PROGRAM pouStation1
VAR
	stationMode: FB_Mode;
	tCalcNumberOfPages: REAL;
	ceil: REAL;
	PartBuild: FB_PartBuild;
	retvall: UDINT;
	
	
	// TODO
	tPartPresent: BOOL;
END_VAR

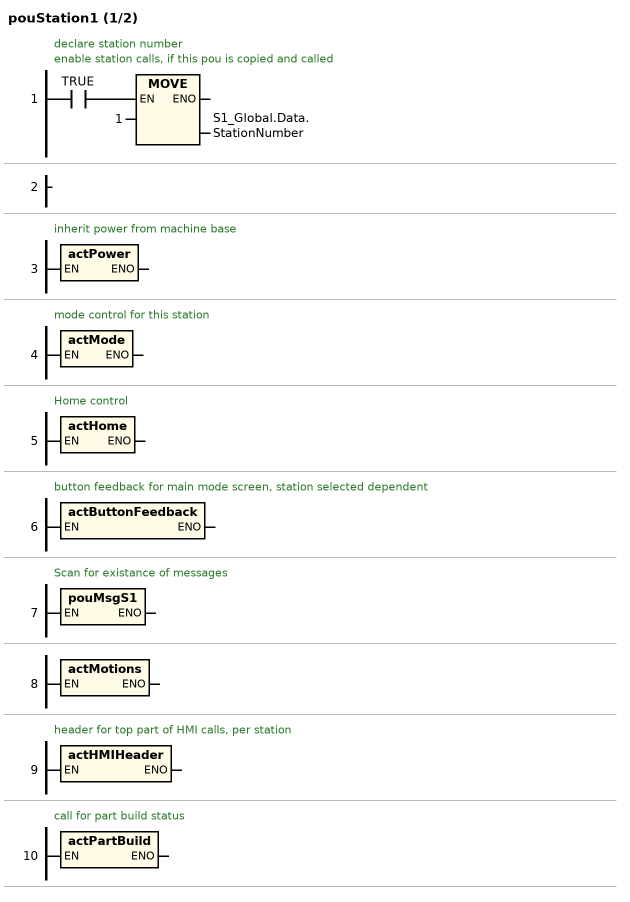
// NETWORK 1
// declare station number
// enable station calls, if this pou is copied and called
S1_Global.Data.StationNumber := 1;

// NETWORK 2

// NETWORK 3
// inherit power from machine base
actPower();

// NETWORK 4
// mode control for this station
actMode();

// NETWORK 5
// Home control
actHome();

// NETWORK 6
// button feedback for main mode screen, station selected dependent
actButtonFeedback();

// NETWORK 7
// Scan for existance of messages
pouMsgS1();

// NETWORK 8
actMotions();

// NETWORK 9
// header for top part of HMI calls, per station
actHMIHeader();

// NETWORK 10
// call for part build status
actPartBuild();

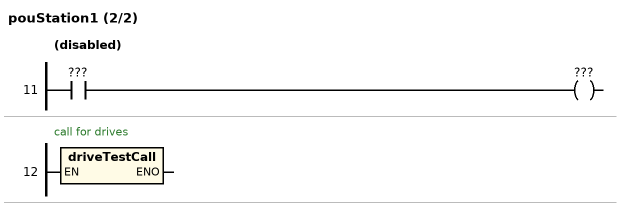
// NETWORK 11 (disabled)
// ??? := ???;

// NETWORK 12
// call for drives
driveTestCall();

ACTION actButtonFeedback:
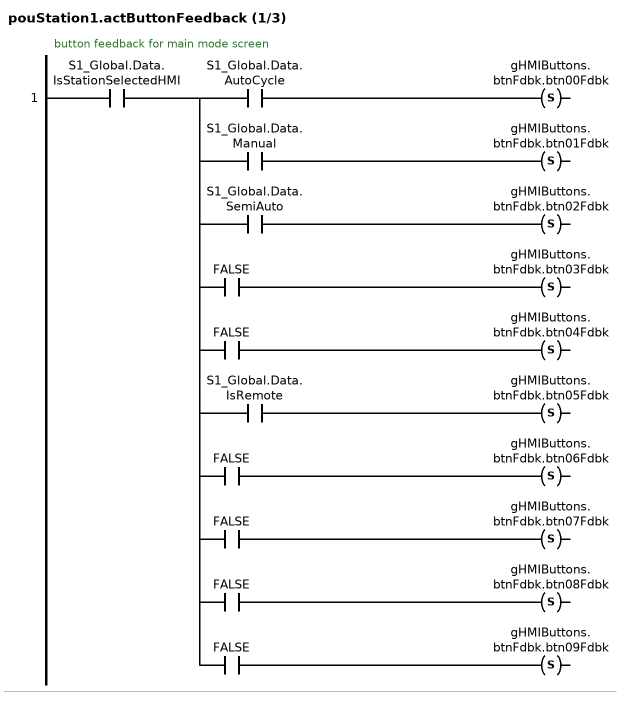
// NETWORK 1
// button feedback for main mode screen
gHMIButtons.btnFdbk.btn00Fdbk S= S1_Global.Data.IsStationSelectedHMI AND S1_Global.Data.AutoCycle;
gHMIButtons.btnFdbk.btn01Fdbk S= S1_Global.Data.IsStationSelectedHMI AND S1_Global.Data.Manual;
gHMIButtons.btnFdbk.btn02Fdbk S= S1_Global.Data.IsStationSelectedHMI AND S1_Global.Data.SemiAuto;
gHMIButtons.btnFdbk.btn03Fdbk S= S1_Global.Data.IsStationSelectedHMI AND FALSE;
gHMIButtons.btnFdbk.btn04Fdbk S= S1_Global.Data.IsStationSelectedHMI AND FALSE;
gHMIButtons.btnFdbk.btn05Fdbk S= S1_Global.Data.IsStationSelectedHMI AND S1_Global.Data.IsRemote;
gHMIButtons.btnFdbk.btn06Fdbk S= S1_Global.Data.IsStationSelectedHMI AND FALSE;
gHMIButtons.btnFdbk.btn07Fdbk S= S1_Global.Data.IsStationSelectedHMI AND FALSE;
gHMIButtons.btnFdbk.btn08Fdbk S= S1_Global.Data.IsStationSelectedHMI AND FALSE;
gHMIButtons.btnFdbk.btn09Fdbk S= S1_Global.Data.IsStationSelectedHMI AND FALSE;

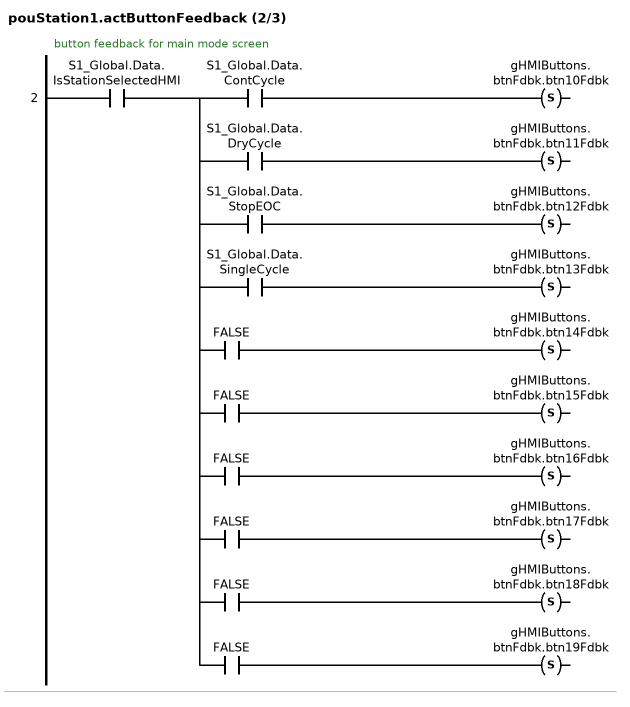
// NETWORK 2
// button feedback for main mode screen
gHMIButtons.btnFdbk.btn10Fdbk S= S1_Global.Data.IsStationSelectedHMI AND S1_Global.Data.ContCycle;
gHMIButtons.btnFdbk.btn11Fdbk S= S1_Global.Data.IsStationSelectedHMI AND S1_Global.Data.DryCycle;
gHMIButtons.btnFdbk.btn12Fdbk S= S1_Global.Data.IsStationSelectedHMI AND S1_Global.Data.StopEOC;
gHMIButtons.btnFdbk.btn13Fdbk S= S1_Global.Data.IsStationSelectedHMI AND S1_Global.Data.SingleCycle;
gHMIButtons.btnFdbk.btn14Fdbk S= S1_Global.Data.IsStationSelectedHMI AND FALSE;
gHMIButtons.btnFdbk.btn15Fdbk S= S1_Global.Data.IsStationSelectedHMI AND FALSE;
gHMIButtons.btnFdbk.btn16Fdbk S= S1_Global.Data.IsStationSelectedHMI AND FALSE;
gHMIButtons.btnFdbk.btn17Fdbk S= S1_Global.Data.IsStationSelectedHMI AND FALSE;
gHMIButtons.btnFdbk.btn18Fdbk S= S1_Global.Data.IsStationSelectedHMI AND FALSE;
gHMIButtons.btnFdbk.btn19Fdbk S= S1_Global.Data.IsStationSelectedHMI AND FALSE;

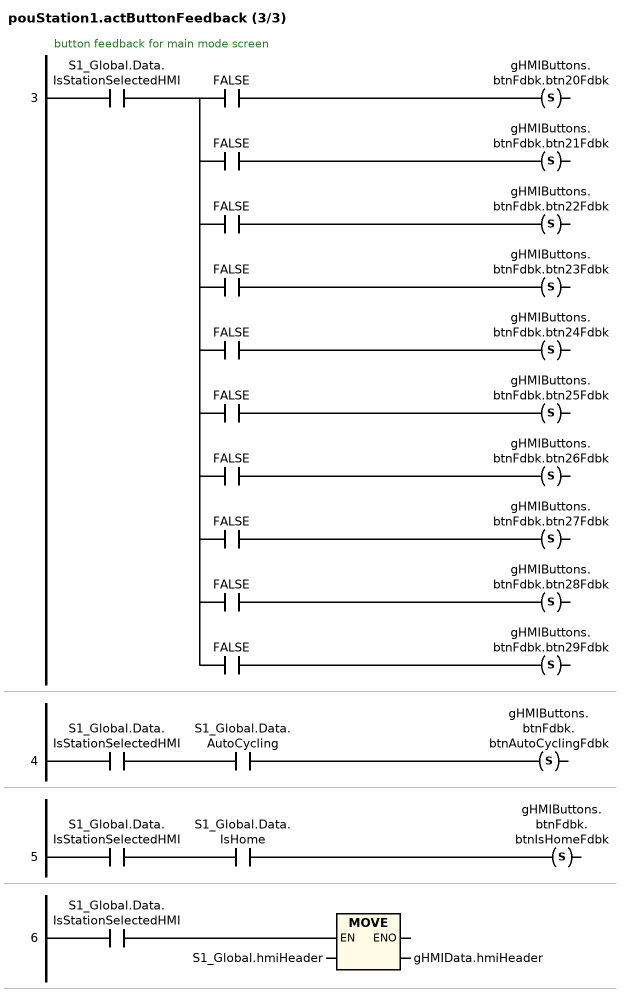
// NETWORK 3
// button feedback for main mode screen
gHMIButtons.btnFdbk.btn20Fdbk S= S1_Global.Data.IsStationSelectedHMI AND FALSE;
gHMIButtons.btnFdbk.btn21Fdbk S= S1_Global.Data.IsStationSelectedHMI AND FALSE;
gHMIButtons.btnFdbk.btn22Fdbk S= S1_Global.Data.IsStationSelectedHMI AND FALSE;
gHMIButtons.btnFdbk.btn23Fdbk S= S1_Global.Data.IsStationSelectedHMI AND FALSE;
gHMIButtons.btnFdbk.btn24Fdbk S= S1_Global.Data.IsStationSelectedHMI AND FALSE;
gHMIButtons.btnFdbk.btn25Fdbk S= S1_Global.Data.IsStationSelectedHMI AND FALSE;
gHMIButtons.btnFdbk.btn26Fdbk S= S1_Global.Data.IsStationSelectedHMI AND FALSE;
gHMIButtons.btnFdbk.btn27Fdbk S= S1_Global.Data.IsStationSelectedHMI AND FALSE;
gHMIButtons.btnFdbk.btn28Fdbk S= S1_Global.Data.IsStationSelectedHMI AND FALSE;
gHMIButtons.btnFdbk.btn29Fdbk S= S1_Global.Data.IsStationSelectedHMI AND FALSE;

// NETWORK 4
gHMIButtons.btnFdbk.btnAutoCyclingFdbk S= S1_Global.Data.IsStationSelectedHMI AND S1_Global.Data.AutoCycling;

// NETWORK 5
gHMIButtons.btnFdbk.btnIsHomeFdbk S= S1_Global.Data.IsStationSelectedHMI AND S1_Global.Data.IsHome;

// NETWORK 6
IF S1_Global.Data.IsStationSelectedHMI THEN gHMIData.hmiHeader := S1_Global.hmiHeader; END_IF
END_ACTION

ACTION actHMIHeader:
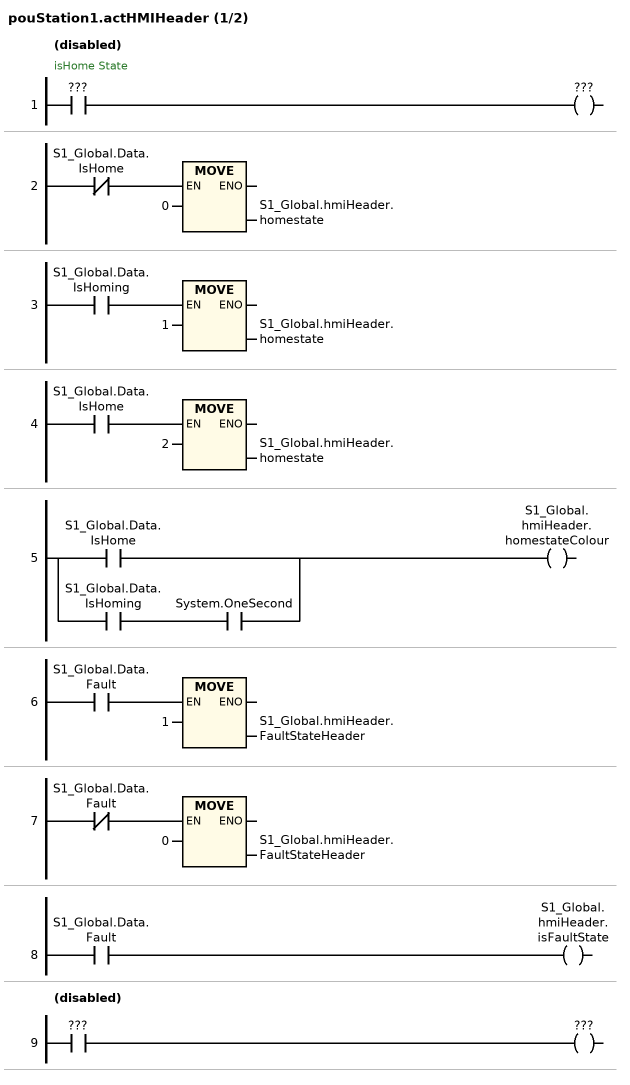
// NETWORK 1 (disabled)
// isHome State
// ??? := ???;

// NETWORK 2
IF NOT S1_Global.Data.IsHome THEN S1_Global.hmiHeader.homestate := 0; END_IF

// NETWORK 3
IF S1_Global.Data.IsHoming THEN S1_Global.hmiHeader.homestate := 1; END_IF

// NETWORK 4
IF S1_Global.Data.IsHome THEN S1_Global.hmiHeader.homestate := 2; END_IF

// NETWORK 5
S1_Global.hmiHeader.homestateColour := S1_Global.Data.IsHome OR S1_Global.Data.IsHoming AND System.OneSecond;

// NETWORK 6
IF S1_Global.Data.Fault THEN S1_Global.hmiHeader.FaultStateHeader := 1; END_IF

// NETWORK 7
IF NOT S1_Global.Data.Fault THEN S1_Global.hmiHeader.FaultStateHeader := 0; END_IF

// NETWORK 8
S1_Global.hmiHeader.isFaultState := S1_Global.Data.Fault;

// NETWORK 9 (disabled)
// ??? := ???;

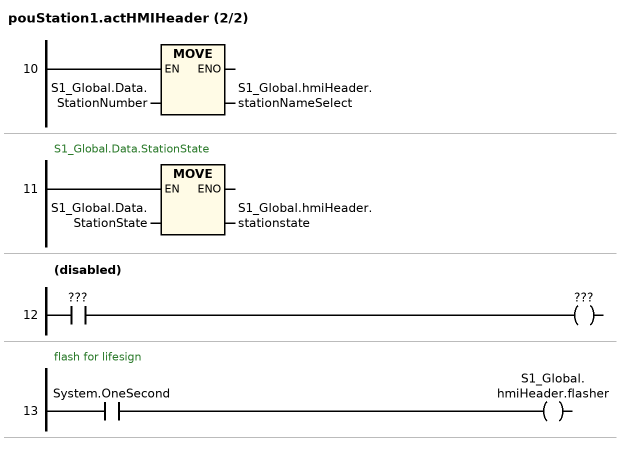
// NETWORK 10
S1_Global.hmiHeader.stationNameSelect := S1_Global.Data.StationNumber;

// NETWORK 11
// S1_Global.Data.StationState
S1_Global.hmiHeader.stationstate := S1_Global.Data.StationState;

// NETWORK 12 (disabled)
// ??? := ???;

// NETWORK 13
// flash for lifesign
S1_Global.hmiHeader.flasher := System.OneSecond;
END_ACTION

ACTION actHome:
//Set home status for station

IF 
//are all motions returned
S1_01_Motion_01_01.Motion.qReturnDepth AND
S1_01_Motion_01_02.Motion.qReturnDepth AND
S1_01_Motion_01_03.Motion.qReturnDepth AND
S1_01_Motion_01_04.Motion.qReturnDepth AND
S1_01_Motion_01_05.Motion.qReturnDepth AND
S1_01_Motion_01_06.Motion.qReturnDepth

	THEN
		//set IsHome value for station
		S1_Global.Data.IsHome := TRUE;
	ELSE
		S1_Global.Data.IsHome := FALSE;
END_IF
END_ACTION

ACTION actMaxNumStationPages:
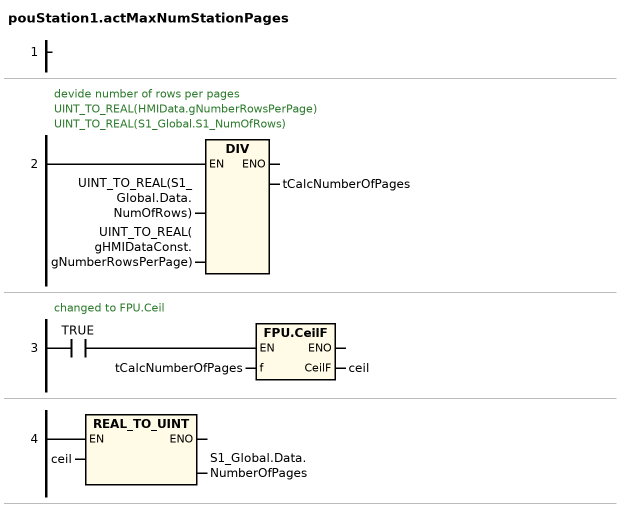
// NETWORK 1

// NETWORK 2
// devide number of rows per pages
// UINT_TO_REAL(HMIData.gNumberRowsPerPage)
// UINT_TO_REAL(S1_Global.S1_NumOfRows)
tCalcNumberOfPages := (UINT_TO_REAL(S1_Global.Data.NumOfRows)) / (UINT_TO_REAL(gHMIDataConst.gNumberRowsPerPage));

// NETWORK 3
// changed to FPU.Ceil
ceil := FPU.CeilF(f := tCalcNumberOfPages);

// NETWORK 4
S1_Global.Data.NumberOfPages := REAL_TO_UINT(ceil);
END_ACTION

ACTION actMode:
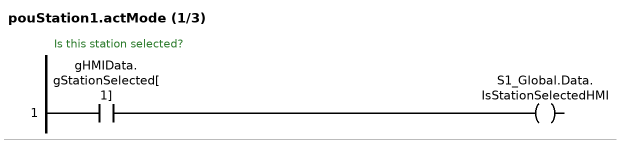
// NETWORK 1
// Is this station selected?
S1_Global.Data.IsStationSelectedHMI := gHMIData.gStationSelected[1];

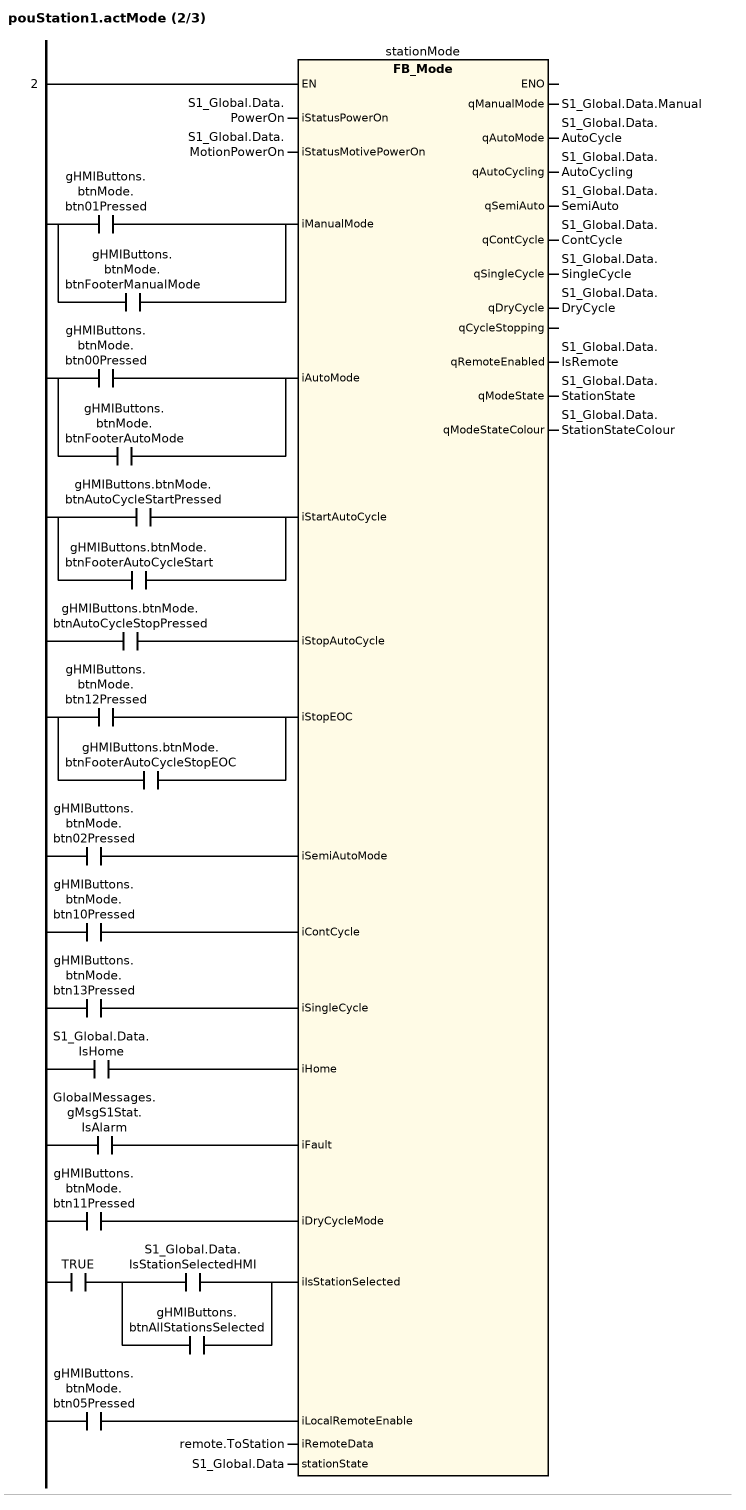
// NETWORK 2
stationMode(
    iStatusPowerOn := S1_Global.Data.PowerOn,
    iStatusMotivePowerOn := S1_Global.Data.MotionPowerOn,
    iManualMode := gHMIButtons.btnMode.btn01Pressed OR gHMIButtons.btnMode.btnFooterManualMode,
    iAutoMode := gHMIButtons.btnMode.btn00Pressed OR gHMIButtons.btnMode.btnFooterAutoMode,
    iStartAutoCycle := gHMIButtons.btnMode.btnAutoCycleStartPressed OR gHMIButtons.btnMode.btnFooterAutoCycleStart,
    iStopAutoCycle := gHMIButtons.btnMode.btnAutoCycleStopPressed,
    iStopEOC := gHMIButtons.btnMode.btn12Pressed OR gHMIButtons.btnMode.btnFooterAutoCycleStopEOC,
    iSemiAutoMode := gHMIButtons.btnMode.btn02Pressed,
    iContCycle := gHMIButtons.btnMode.btn10Pressed,
    iSingleCycle := gHMIButtons.btnMode.btn13Pressed,
    iHome := S1_Global.Data.IsHome,
    iFault := GlobalMessages.gMsgS1Stat.IsAlarm,
    iDryCycleMode := gHMIButtons.btnMode.btn11Pressed,
    iIsStationSelected := TRUE AND (S1_Global.Data.IsStationSelectedHMI OR gHMIButtons.btnAllStationsSelected),
    iLocalRemoteEnable := gHMIButtons.btnMode.btn05Pressed,
    iRemoteData := remote.ToStation,
    stationState := S1_Global.Data,
    qManualMode => S1_Global.Data.Manual,
    qAutoMode => S1_Global.Data.AutoCycle,
    qAutoCycling => S1_Global.Data.AutoCycling,
    qSemiAuto => S1_Global.Data.SemiAuto,
    qContCycle => S1_Global.Data.ContCycle,
    qSingleCycle => S1_Global.Data.SingleCycle,
    qDryCycle => S1_Global.Data.DryCycle,
    qRemoteEnabled => S1_Global.Data.IsRemote,
    qModeState => S1_Global.Data.StationState,
    qModeStateColour => S1_Global.Data.StationStateColour); // FB_Mode

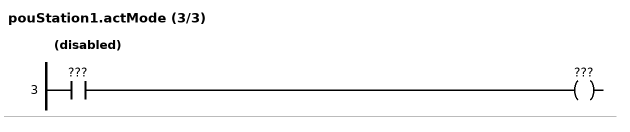
// NETWORK 3 (disabled)
// ??? := ???;
END_ACTION

ACTION actMotions:
//station 1 = 10000 index


//init number of rows
S1_Global.Data.NumOfRows := 0;

//page 1
S1_01_Motion_01_01();
S1_01_Motion_01_02();
S1_01_Motion_01_03();
S1_01_Motion_01_04();
S1_01_Motion_01_05();
S1_01_Motion_01_06();

//page 2
S1_01_Motion_02_07();
S1_01_Motion_02_08();
S1_01_Motion_02_09();
S1_01_Motion_02_10();
S1_01_Motion_02_11();
S1_01_Motion_02_12();

//page 3
S1_01_Motion_03_13();
S1_01_Motion_03_14();
S1_01_Motion_03_15();
S1_01_Motion_03_16();
S1_01_Motion_03_17();
S1_01_Motion_03_18();

//page 4
S1_01_Motion_04_19();
S1_01_Motion_04_20();
S1_01_Motion_04_21();
S1_01_Motion_04_22();
S1_01_Motion_04_23();
S1_01_Motion_04_24();

//page 5
S1_01_Motion_05_25();
S1_01_Motion_05_26();
S1_01_Motion_05_27();
S1_01_Motion_05_28();
S1_01_Motion_05_29();
S1_01_Motion_05_30();

//page 6
S1_01_Motion_06_31();
S1_01_Motion_06_32();
S1_01_Motion_06_33();
S1_01_Motion_06_34();
S1_01_Motion_06_35();
S1_01_Motion_06_36();

//must be called after motionRow calls
actMaxNumStationPages();
END_ACTION

ACTION actPartBuild:
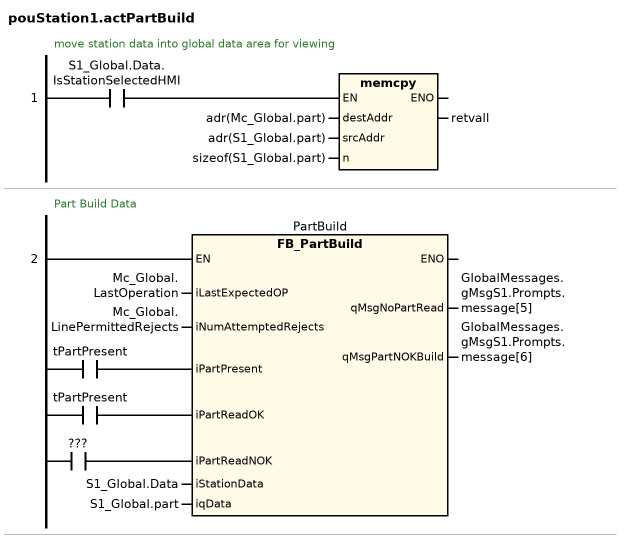
// NETWORK 1
// move station data into global data area for viewing
IF S1_Global.Data.IsStationSelectedHMI THEN
    retvall := memcpy(destAddr := adr(Mc_Global.part), srcAddr := adr(S1_Global.part), n := sizeof(S1_Global.part));
END_IF

// NETWORK 2
// Part Build Data
PartBuild(
    iLastExpectedOP := Mc_Global.LastOperation,
    iNumAttemptedRejects := Mc_Global.LinePermittedRejects,
    iPartPresent := tPartPresent,
    iPartReadOK := tPartPresent,
    iStationData := S1_Global.Data,
    iqData := S1_Global.part,
    qMsgNoPartRead => GlobalMessages.gMsgS1.Prompts.message[5],
    qMsgPartNOKBuild => GlobalMessages.gMsgS1.Prompts.message[6]); // FB_PartBuild
END_ACTION

ACTION actPower:
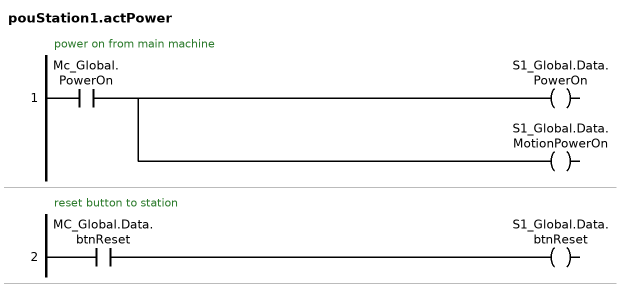
// NETWORK 1
// power on from main machine
S1_Global.Data.PowerOn := Mc_Global.PowerOn;
S1_Global.Data.MotionPowerOn := Mc_Global.PowerOn;

// NETWORK 2
// reset button to station
S1_Global.Data.btnReset := MC_Global.Data.btnReset;
END_ACTION

END_PROGRAM

(* stored: Version 1.1.0.1, ProductVersion 3.1.4024.12
   POU pouStation1: Id {cbb126a5-ed47-44bc-850e-38b5e1137b4b}, SpecialFunc None
   Action actButtonFeedback: Id {346b2711-253c-4729-8cdf-c7e225583299}
   Action actHMIHeader: Id {a5642540-d8e2-4c19-baff-767dcd8b3693}
   Action actHome: Id {38f1ab27-9e47-4a19-9a7c-14bf7a049522}
   Action actMaxNumStationPages: Id {499acf2e-11f1-41ab-acd8-6d6b219bcc13}
   Action actMode: Id {9732a77c-e29b-4611-92cd-047d0b53dcd5}
   Action actMotions: Id {e014ca83-598c-489c-8352-44bf4d8deaf0}
   Action actPartBuild: Id {e298ac78-2bd3-48b2-9423-2952ffbdc450}
   Action actPower: Id {ccf151c7-3331-4fe7-aca1-44f65b2a812b} *)
